PROGRAM P_CounterTest
VAR
	i: INT := 0;
END_VAR

(* Counter just to use memory *)

i := i+1;
IF i >= 65535 THEN
	i := 0;
END_IF

END_PROGRAM

(* stored: Version 1.1.0.1, ProductVersion 3.1.4024.12
   POU P_CounterTest: Id {2425c3ab-e7fe-4c29-818b-039c06e0d523}, SpecialFunc None *)
